# EPICS autosave request: vme_iocs/iocbio4/iocBoot/ioc18IDd/auto_settings.req
# Note: the macro P must have been supplied to the routine that parses
# this file.  Normally, this means a command like the following is in st.cmd
# create_monitor_set("auto_settings.req",30,"P=18IDd:")
# This requires save_restore v2.8 or later.

#file softMotor_settings.req P=$(P),SM=SM1
#file softMotor_settings.req P=$(P),SM=SM2
#file softMotor_settings.req P=$(P),SM=SM3
#file softMotor_settings.req P=$(P),SM=SM4
#file softMotor_settings.req P=$(P),SM=SM5
#file softMotor_settings.req P=$(P),SM=SM6
#file softMotor_settings.req P=$(P),SM=SM7
#file softMotor_settings.req P=$(P),SM=SM8
#file softMotor_settings.req P=$(P),SM=SM9
#file softMotor_settings.req P=$(P),SM=SM10

file scaler_8ch_settings.req P=$(P)mcs:,S=scaler1

file scan_settings.req P=$(P),S=scan1
file scan_settings.req P=$(P),S=scan2
file scan_settings.req P=$(P),S=scan3
file scan_settings.req P=$(P),S=scan4
file scan_settings.req P=$(P),S=scanH
file saveData_settings.req P=$(P)

# Kohzu monochromator
#file kohzuSeq_settings.req P=$(P)

# High resolution monochromator
#file hrSeq_settings.req P=$(P),N=1

# Io calc
#file Io_settings.req P=18IDd:Io:

#$(P)fltr1:name5.VAL
#$(P)fltr1:name4.VAL
#$(P)fltr1:name3.VAL
#$(P)fltr1:name2.VAL
#$(P)fltr1:name1.VAL
#$(P)fltr1:nameHome.VAL
#$(P)fltr1:pos5.VAL
#$(P)fltr1:pos4.VAL
#$(P)fltr1:pos3.VAL
#$(P)fltr1:pos2.VAL
#$(P)fltr1:pos1.VAL
#$(P)fltr1:posHome.VAL
#$(P)fltr1:motorOut.OUTN
#$(P)fltr2:name5.VAL
#$(P)fltr2:name4.VAL
#$(P)fltr2:name3.VAL
#$(P)fltr2:name2.VAL
#$(P)fltr2:name1.VAL
#$(P)fltr2:nameHome.VAL
#$(P)fltr2:pos5.VAL
#$(P)fltr2:pos4.VAL
#$(P)fltr2:pos3.VAL
#$(P)fltr2:pos2.VAL
#$(P)fltr2:pos1.VAL
#$(P)fltr2:posHome.VAL
#$(P)fltr2:motorOut.OUTN
#$(P)fltr_1_2:lockOut.OUTN

file userCalcs10_settings.req P=$(P)
#$(P)userCalcEnable.VAL

file userTransforms10_settings.req P=$(P)
#$(P)userTranEnable.VAL

file userStringCalcs10_settings.req P=$(P)
#$(P)userStringCalcEnable.VAL

file userStringSeqs10_settings.req P=$(P)
#$(P)userStringSeqEnable

file userArrayCalcs10_settings.req P=$(P)
#$(P)userArrayCalcEnable.VAL

# 4-step measurement
file auto_4step_settings.req P=$(P),Q=4step

file userAve10_settings.req P=$(P)
$(P)userAveEnable.VAL

file interp_settings.req P=$(P)

# MCA
#file mca_settings.req P=$(P),M=aim_adc1
#file icb_adc_settings.req P=$(P),ADC=adc1
#file icb_amp_settings.req P=$(P),AMP=amp1
#file icb_hvps_settings.req P=$(P),HVPS=hvps1
#file icb_tca_settings.req P=$(P),TCA=tca1
#file icbDsp_settings.req P=$(P),DSP=dsp1

# orientation matrix
#file orient_settings.req P=$(P),O=1
#file orient_xtals_settings.req P=$(P),O=1

# pvHistory
#file pvHistory.req P=$(P),N=1

#file CoarseFineMotor_settings.req P=18IDd:cf1:

# XIA slit
#$(P)hsc1:hID
#$(P)hsc1:vID
#$(P)hsc1:enable
#$(P)hsc1:debug

## Femto amplifier 4
#file femto.req P=$(P),H=fem01:,F=seq01:

## PF4 dual filter
#file pf4dual.req P=$(P),H=pf401:,F=seq01:

#file deviceCmdReply.req P=$(P),N=1

#file timer.req P=$(P),N=1
file k428_settings.req P=18ID:,M=k428-10:
file k428_settings.req P=18ID:,M=k428-11:
file k428_settings.req P=18ID:,M=k428-12:
file k428_settings.req P=18ID:,M=k428-13:
